# EPICS autosave request: iocBoot/generic_motors_ioc/dbSave/XY_P3_.req
%
% BURT Request File
%
% $(P)XY:P3:  X-Y positioner #3
%

file assy.req ASSY=$(P)XY:P3
file mtr1.req MTR1=$(P)XY:mx3
file mtr1.req MTR1=$(P)XY:my3
file drv1.req DRV1=$(P)XY:X3
file drv1.req DRV1=$(P)XY:Y3
